// TIA Portal V16 export
// export: Created 2024-09-05T17:39:14.0932833Z, ExportSetting WithDefaults, DisplayName Totally Integrated Automation Portal, DisplayVersion V16 Update 6, DisplayName TIA Portal Version Control Interface, DisplayVersion V16 Update 2, DisplayName TIA Portal Openness, DisplayVersion V16 Update 6, DisplayName STEP 7 Professional, DisplayVersion V16 Update 6, DisplayName STEP 7 Safety, DisplayVersion V16, DisplayName WinCC Advanced, DisplayVersion V16 Update 6
DATA_BLOCK "Manual_DB"   // DB53
VERSION : 0.1
// stored: AutoNumber true, DBAccessibleFromOPCUA true, InstanceOfName Manual, InstanceOfType FB
"Manual"
   // VAR
   //    res : Bool := FALSE;
   //    R_TRIG_MM220bp { S7_SetPoint := 'True'} : R_TRIG;
   //    R_TRIG_MM220wp { S7_SetPoint := 'True'} : R_TRIG;
   //    R_TRIG_MM222bp { S7_SetPoint := 'True'} : R_TRIG;
   //    R_TRIG_MM222wp { S7_SetPoint := 'True'} : R_TRIG;
   //    R_TRIG_MM224bp { S7_SetPoint := 'True'} : R_TRIG;
   //    R_TRIG_MM224wp { S7_SetPoint := 'True'} : R_TRIG;
   // END_VAR
BEGIN
   R_TRIG_MM220bp.CLK := FALSE;
   R_TRIG_MM220bp.Q := FALSE;
   R_TRIG_MM220bp.Stat_Bit := FALSE;
   R_TRIG_MM220wp.CLK := FALSE;
   R_TRIG_MM220wp.Q := FALSE;
   R_TRIG_MM220wp.Stat_Bit := FALSE;
   R_TRIG_MM222bp.CLK := FALSE;
   R_TRIG_MM222bp.Q := FALSE;
   R_TRIG_MM222bp.Stat_Bit := FALSE;
   R_TRIG_MM222wp.CLK := FALSE;
   R_TRIG_MM222wp.Q := FALSE;
   R_TRIG_MM222wp.Stat_Bit := FALSE;
   R_TRIG_MM224bp.CLK := FALSE;
   R_TRIG_MM224bp.Q := FALSE;
   R_TRIG_MM224bp.Stat_Bit := FALSE;
   R_TRIG_MM224wp.CLK := FALSE;
   R_TRIG_MM224wp.Q := FALSE;
   R_TRIG_MM224wp.Stat_Bit := FALSE;
END_DATA_BLOCK
